% RSLogix 500 project Sesion9_Tarea1_Josue Santana Robledo Corona.RSS, saved by version 8.40.00.08 %
PROJECT "UNTITLED"    % processor: MicroLogix 1200 %

PROGRAM FILES
  LAD 2 "MAIN"  4 rungs
  LAD 3 "ENTRADAS"  12 rungs
  LAD 4 "SALIDAS"  5 rungs
  LAD 5 "AUTOMATICO"  10 rungs
  LAD 6 "ALARMAS"  1 rungs
  LAD 7 "HMI"  1 rungs
  LAD 8 "MANUAL"  1 rungs

DATA FILES
  O0 OUTPUT  4 elements
  I1 INPUT  4 elements
  S2 STATUS  66 elements
  B3 BINARY  2 elements
  T4 TIMER  1 elements
  C5 COUNTER  1 elements
  R6 CONTROL  1 elements
  N7 INTEGER  1 elements
  F8 FLOAT  1 elements

LADDER 2 "MAIN"
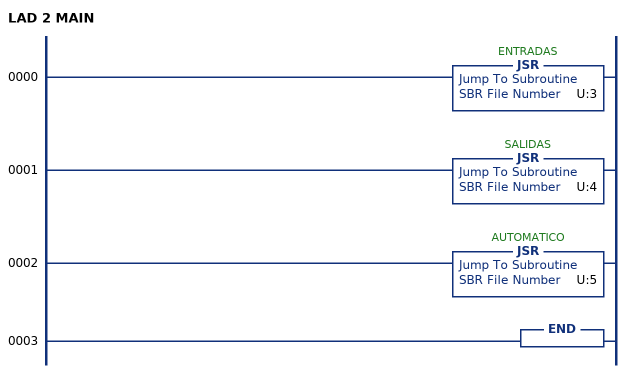
% Rung: 0 %
SOR JSR U:3 EOR
%   U:3  ENTRADAS %
% Rung: 1 %
SOR JSR U:4 EOR
%   U:4  SALIDAS %
% Rung: 2 %
SOR JSR U:5 EOR
%   U:5  AUTOMATICO %
% Rung: 3 %
SOR END EOR

LADDER 3 "ENTRADAS"
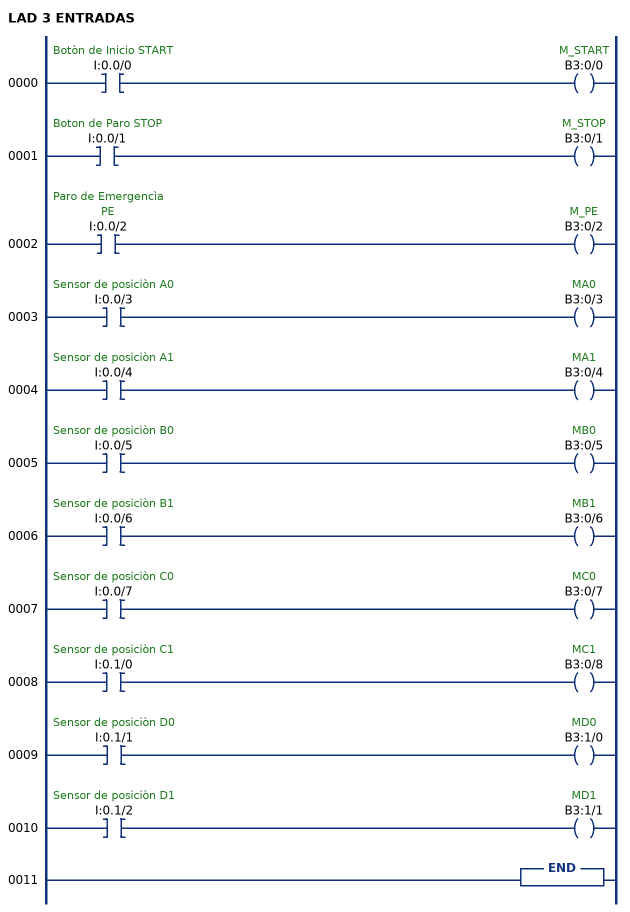
% Rung: 0 %
SOR XIC I:0.0/0 OTE B3:0/0 EOR
%   I:0.0/0  START  "Botòn de Inicio" %
%   B3:0/0  M_START %
% Rung: 1 %
SOR XIC I:0.0/1 OTE B3:0/1 EOR
%   I:0.0/1  STOP  "Boton de Paro" %
%   B3:0/1  M_STOP %
% Rung: 2 %
SOR XIC I:0.0/2 OTE B3:0/2 EOR
%   I:0.0/2  PE  "Paro de Emergencìa" %
%   B3:0/2  M_PE %
% Rung: 3 %
SOR XIC I:0.0/3 OTE B3:0/3 EOR
%   I:0.0/3  A0  "Sensor de posiciòn" %
%   B3:0/3  MA0 %
% Rung: 4 %
SOR XIC I:0.0/4 OTE B3:0/4 EOR
%   I:0.0/4  A1  "Sensor de posiciòn" %
%   B3:0/4  MA1 %
% Rung: 5 %
SOR XIC I:0.0/5 OTE B3:0/5 EOR
%   I:0.0/5  B0  "Sensor de posiciòn" %
%   B3:0/5  MB0 %
% Rung: 6 %
SOR XIC I:0.0/6 OTE B3:0/6 EOR
%   I:0.0/6  B1  "Sensor de posiciòn" %
%   B3:0/6  MB1 %
% Rung: 7 %
SOR XIC I:0.0/7 OTE B3:0/7 EOR
%   I:0.0/7  C0  "Sensor de posiciòn" %
%   B3:0/7  MC0 %
% Rung: 8 %
SOR XIC I:0.1/0 OTE B3:0/8 EOR
%   I:0.1/0  C1  "Sensor de posiciòn" %
%   B3:0/8  MC1 %
% Rung: 9 %
SOR XIC I:0.1/1 OTE B3:1/0 EOR
%   I:0.1/1  D0  "Sensor de posiciòn" %
%   B3:1/0  MD0 %
% Rung: 10 %
SOR XIC I:0.1/2 OTE B3:1/1 EOR
%   I:0.1/2  D1  "Sensor de posiciòn" %
%   B3:1/1  MD1 %
% Rung: 11 %
SOR END EOR

LADDER 4 "SALIDAS"
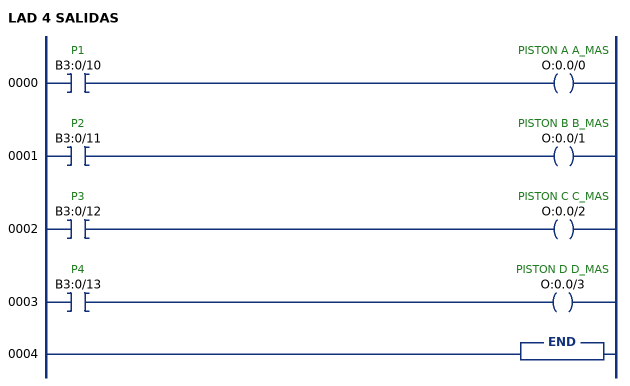
% Rung: 0 %
SOR XIC B3:0/10 OTE O:0.0/0 EOR
%   B3:0/10  P1 %
%   O:0.0/0  A_MAS  "PISTON A" %
% Rung: 1 %
SOR XIC B3:0/11 OTE O:0.0/1 EOR
%   B3:0/11  P2 %
%   O:0.0/1  B_MAS  "PISTON B" %
% Rung: 2 %
SOR XIC B3:0/12 OTE O:0.0/2 EOR
%   B3:0/12  P3 %
%   O:0.0/2  C_MAS  "PISTON C" %
% Rung: 3 %
SOR XIC B3:0/13 OTE O:0.0/3 EOR
%   B3:0/13  P4 %
%   O:0.0/3  D_MAS  "PISTON D" %
% Rung: 4 %
SOR END EOR

LADDER 5 "AUTOMATICO"
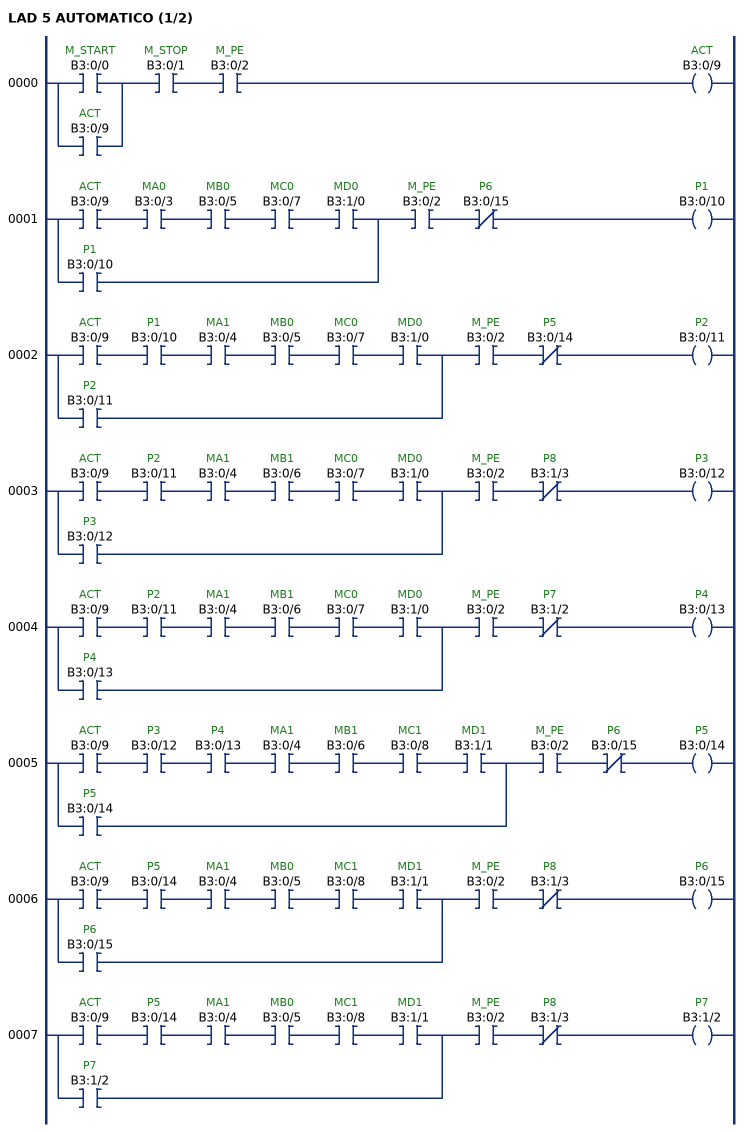
% Rung: 0 %
SOR BST XIC B3:0/0 NXB XIC B3:0/9 BND XIC B3:0/1 XIC B3:0/2 OTE B3:0/9 EOR
%   B3:0/0  M_START %
%   B3:0/9  ACT %
%   B3:0/1  M_STOP %
%   B3:0/2  M_PE %
% Rung: 1 %
SOR BST XIC B3:0/9 XIC B3:0/3 XIC B3:0/5 XIC B3:0/7 XIC B3:1/0 NXB XIC B3:0/10 BND XIC B3:0/2 XIO B3:0/15 OTE B3:0/10 EOR
%   B3:0/9  ACT %
%   B3:0/3  MA0 %
%   B3:0/5  MB0 %
%   B3:0/7  MC0 %
%   B3:1/0  MD0 %
%   B3:0/10  P1 %
%   B3:0/2  M_PE %
%   B3:0/15  P6 %
% Rung: 2 %
SOR BST XIC B3:0/9 XIC B3:0/10 XIC B3:0/4 XIC B3:0/5 XIC B3:0/7 XIC B3:1/0 NXB XIC B3:0/11 BND XIC B3:0/2 XIO B3:0/14 OTE B3:0/11 EOR
%   B3:0/9  ACT %
%   B3:0/10  P1 %
%   B3:0/4  MA1 %
%   B3:0/5  MB0 %
%   B3:0/7  MC0 %
%   B3:1/0  MD0 %
%   B3:0/11  P2 %
%   B3:0/2  M_PE %
%   B3:0/14  P5 %
% Rung: 3 %
SOR BST XIC B3:0/9 XIC B3:0/11 XIC B3:0/4 XIC B3:0/6 XIC B3:0/7 XIC B3:1/0 NXB XIC B3:0/12 BND XIC B3:0/2 XIO B3:1/3 OTE B3:0/12 EOR
%   B3:0/9  ACT %
%   B3:0/11  P2 %
%   B3:0/4  MA1 %
%   B3:0/6  MB1 %
%   B3:0/7  MC0 %
%   B3:1/0  MD0 %
%   B3:0/12  P3 %
%   B3:0/2  M_PE %
%   B3:1/3  P8 %
% Rung: 4 %
SOR BST XIC B3:0/9 XIC B3:0/11 XIC B3:0/4 XIC B3:0/6 XIC B3:0/7 XIC B3:1/0 NXB XIC B3:0/13 BND XIC B3:0/2 XIO B3:1/2 OTE B3:0/13 EOR
%   B3:0/9  ACT %
%   B3:0/11  P2 %
%   B3:0/4  MA1 %
%   B3:0/6  MB1 %
%   B3:0/7  MC0 %
%   B3:1/0  MD0 %
%   B3:0/13  P4 %
%   B3:0/2  M_PE %
%   B3:1/2  P7 %
% Rung: 5 %
SOR BST XIC B3:0/9 XIC B3:0/12 XIC B3:0/13 XIC B3:0/4 XIC B3:0/6 XIC B3:0/8 XIC B3:1/1 NXB XIC B3:0/14 BND XIC B3:0/2 XIO B3:0/15 OTE B3:0/14 EOR
%   B3:0/9  ACT %
%   B3:0/12  P3 %
%   B3:0/13  P4 %
%   B3:0/4  MA1 %
%   B3:0/6  MB1 %
%   B3:0/8  MC1 %
%   B3:1/1  MD1 %
%   B3:0/14  P5 %
%   B3:0/2  M_PE %
%   B3:0/15  P6 %
% Rung: 6 %
SOR BST XIC B3:0/9 XIC B3:0/14 XIC B3:0/4 XIC B3:0/5 XIC B3:0/8 XIC B3:1/1 NXB XIC B3:0/15 BND XIC B3:0/2 XIO B3:1/3 OTE B3:0/15 EOR
%   B3:0/9  ACT %
%   B3:0/14  P5 %
%   B3:0/4  MA1 %
%   B3:0/5  MB0 %
%   B3:0/8  MC1 %
%   B3:1/1  MD1 %
%   B3:0/15  P6 %
%   B3:0/2  M_PE %
%   B3:1/3  P8 %
% Rung: 7 %
SOR BST XIC B3:0/9 XIC B3:0/14 XIC B3:0/4 XIC B3:0/5 XIC B3:0/8 XIC B3:1/1 NXB XIC B3:1/2 BND XIC B3:0/2 XIO B3:1/3 OTE B3:1/2 EOR
%   B3:0/9  ACT %
%   B3:0/14  P5 %
%   B3:0/4  MA1 %
%   B3:0/5  MB0 %
%   B3:0/8  MC1 %
%   B3:1/1  MD1 %
%   B3:1/2  P7 %
%   B3:0/2  M_PE %
%   B3:1/3  P8 %

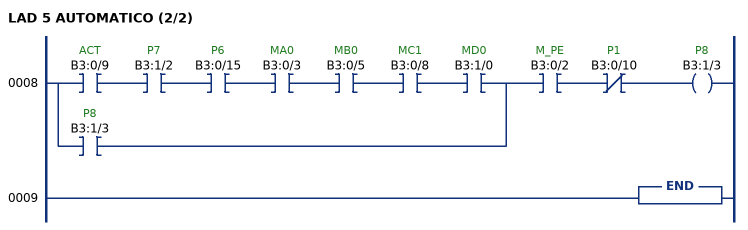
% Rung: 8 %
SOR BST XIC B3:0/9 XIC B3:1/2 XIC B3:0/15 XIC B3:0/3 XIC B3:0/5 XIC B3:0/8 XIC B3:1/0 NXB XIC B3:1/3 BND XIC B3:0/2 XIO B3:0/10 OTE B3:1/3 EOR
%   B3:0/9  ACT %
%   B3:1/2  P7 %
%   B3:0/15  P6 %
%   B3:0/3  MA0 %
%   B3:0/5  MB0 %
%   B3:0/8  MC1 %
%   B3:1/0  MD0 %
%   B3:1/3  P8 %
%   B3:0/2  M_PE %
%   B3:0/10  P1 %
% Rung: 9 %
SOR END EOR
